//********************************************************************************
// FUN_Cartesian to polar.
// -------------------------------------------------------------------------------
// This function calculates the polar coordinates r and theta from
// the cartesian X and Y coordinates. 
//	
// Version:
//			- V1.01	HHL, 11/05-2022
//********************************************************************************
FUNCTION FUN_CartesianToPolar : LREAL
VAR_IN_OUT
END_VAR
VAR_INPUT
	fX				:REAL;			// X-axis coordinate
	fY				:REAL;			// Y-axis coordinate
END_VAR
VAR_OUTPUT
	fRadius			:REAL;			// Radius for polar coordinate
	fAngle			:REAL;			// [deg] Angle for polar coordinate 
END_VAR
VAR
	bError			:BOOL;			// True if error occured during determination of angle
END_VAR


// Calculate polar coordinates from cartesian coordinates
//-----------------------------------------

// Calculate radius
fRadius := LREAL_TO_REAL(SQRT((EXPT(fX,2) + EXPT(fY,2))));

// Calculate angle
IF fX <> 0 THEN 
	// Calculate angle 
	IF 0 <= fX AND 0 <= fY THEN
		// I. Quadrant	
		IF fX <> 0 THEN
			fAngle := LREAL_TO_REAL(RAD_TO_DEG(ATAN(fY/fX)));
		ELSIF fX = 0 THEN
			IF fY > 0 THEN
				fAngle := 90.0;
			ELSIF fY = 0 THEN
				// Special case where both fX and fY are zero.
				bError := TRUE;
			END_IF
		END_IF
	ELSIF 0 > fX AND 0 <= fY THEN 	
		// II. Quadrant	
		IF fY <> 0 THEN
			fAngle := LREAL_TO_REAL(RAD_TO_DEG(ATAN(fY/fX)) + 180);
		ELSIF fY = 0 THEN
			IF fX > 0 THEN
				fAngle := 0.0;
			ELSE
				fAngle := -180.0;
			END_IF
		END_IF
	ELSIF 0 > fX AND 0 > fY THEN 	
		// III. Quadrant	
		fAngle := -1*(180 - LREAL_TO_REAL(RAD_TO_DEG(ATAN(fY/fX))));
	ELSIF 0 < fX AND 0 > fY THEN 	
		// IV. Quadrant	
		fAngle := LREAL_TO_REAL(RAD_TO_DEG(ATAN(fY/fX)));
	END_IF	
ELSE
	// X-axis coordinate is zero 
	IF fY = 0 THEN
		fAngle  := 0.0;		
	ELSIF fY > 0 THEN
		fAngle  := 90.0;
	ELSE
 		fAngle  := -90.0;
	END_IF
END_IF

END_FUNCTION

(* stored: Version 1.1.0.1, ProductVersion 3.1.4024.12
   POU FUN_CartesianToPolar: Id {d48ff7a6-2ca5-42ac-b609-bbcc969cc5c6}, SpecialFunc None *)
